{attribute addProperty BoxType "EK1122-0000-0018"}
{attribute addProperty Id "Beckhoff_APS1xxxsub_EK1100EK1100_179A0949162A_0001_APS1003_7000_0016APS1003_C39F7B892112264"}
{attribute addProperty CRC "1549976076"}
{attribute addProperty SizeInBites "2128"}
{attribute addProperty SizeInBytes "266"}
TYPE Beckhoff_APS1xxxEK1122_5C62C20C EXTENDS EK1122_179A0949 :
STRUCT
	{attribute addProperty Name "Beckhoff_APS1xxxsub_EK1100"}
	Beckhoff_APS1xxxsub_EK1100 : EK1100_179A0949;
	{attribute addProperty Name "A_0001_APS1003_7000_0016"}
	A_0001_APS1003_7000_0016 : APS1003_C39F7B89;
END_STRUCT
END_TYPE

(* stored: Version 1.2.0.0, ProductVersion 3.1.4024.9
   DUT Beckhoff_APS1xxxEK1122_5C62C20C: Id {3890200c-4cfe-44ba-8556-d510245ad9cc} *)
